{attribute 'linkalways'} 
{attribute 'no_explicit_call' := 'This FB is a CLASS and must be accessed using methods or properties'}
{attribute 'enable_dynamic_creation'}
FUNCTION_BLOCK _TcVnArray4_Point2_REAL EXTENDS AliasDatatypeBase
VAR
	localData : TcVnArray4_Point2_REAL;
	activeData : REFERENCE TO TcVnArray4_Point2_REAL REF= localData;
	aliasBaseDatatype : _Array0to3OfTcVnPoint2_REAL;
END_VAR

PROPERTY PUBLIC Address : PVOID
GET
Address := ADR(activeData);
END_GET
END_PROPERTY

METHOD PUBLIC ClearReference
VAR_INPUT
END_VAR
activeData REF= localData;
SetBaseDatatypeReference();
END_METHOD

METHOD PUBLIC Clone : I_Datatype
VAR
    pClone : POINTER TO _TcVnArray4_Point2_REAL;
END_VAR
pClone := __NEW(_TcVnArray4_Point2_REAL);
Clone := pClone^;
END_METHOD

METHOD FB_init : BOOL
VAR_INPUT
	bInitRetains : BOOL; // if TRUE, the retain variables are initialized (warm start / cold start)
	bInCopyCode : BOOL;  // if TRUE, the instance afterwards gets moved into the copy code (online change)
	//InitialValue : TcVnArray4_LREAL; // if possible, not all values can be initialized
END_VAR
//localData := InitialValue; // if possible, not all values can be initialized
SetBaseDatatypeReference();
AddBaseDatatype(aliasBaseDatatype);
END_METHOD

PROPERTY PUBLIC Identifier : T_MAXSTRING
GET
Identifier := 'TcVnArray4_Point2_REAL';
END_GET
END_PROPERTY

METHOD PUBLIC MakeReferenceTo
VAR_INPUT
	ReferenceTarget : REFERENCE TO TcVnArray4_Point2_REAL;
END_VAR
activeData REF= ReferenceTarget;
SetBaseDatatypeReference();
END_METHOD

METHOD PROTECTED SetBaseDatatypeReference
VAR_INPUT
END_VAR
aliasBaseDatatype.MakeReferenceTo(activeData);
END_METHOD

PROPERTY PUBLIC Size : UDINT
GET
Size := SIZEOF(activeData);
END_GET
END_PROPERTY

METHOD TryMakeReferenceTo : BOOL
VAR_INPUT
	Target : I_Datatype;
END_VAR
VAR
	pTargetData : POINTER TO TcVnArray4_Point2_REAL;
END_VAR
IF NOT IsEquivalentTo(Target) THEN
	RETURN;
END_IF

pTargetData := Target.Address;
activeData REF= pTargetData^;
SetBaseDatatypeReference();
TryMakeReferenceTo := TRUE;
END_METHOD

PROPERTY PUBLIC Value : REFERENCE TO TcVnArray4_Point2_REAL
GET
Value REF= activeData;
END_GET
END_PROPERTY

END_FUNCTION_BLOCK

(* stored: Version 1.1.0.1, ProductVersion 3.1.4024.13
   POU _TcVnArray4_Point2_REAL: Id {4025545f-dcd8-07f1-1107-87b0a050a007}, SpecialFunc None
   Folder Core: Id {1c224fdd-c286-067e-04f2-d6bc7c35533d}
   Folder Protected: Id {4b953cbc-0aa4-0180-3702-b88e6c1fe404}
   Folder Customize: Id {2d5a0047-d894-0c0c-1809-63d4316bbc29}
   Folder Constructor: Id {300c001e-6c28-0191-2240-26d28b2c7c34}
   Property Address: Id {fc659714-5bc5-0c7c-387d-10f77cbd39fe}
   Get Get: Id {d3ed5257-1d97-0b2d-1f86-5ac107c9d8f9}
   Method ClearReference: Id {282ccc3b-dbad-0830-2569-5c5e0bd79fea}
   Method Clone: Id {c3c1805b-f6b4-0162-321b-9fd4d2ee7ef1}
   Method FB_init: Id {7e656011-61f9-001c-3cc3-15cd8dc4d22e}
   Property Identifier: Id {87984a0e-07fe-0af7-3a9f-af2a916713fd}
   Get Get: Id {f0e7879e-9d2b-0d16-28fd-4b66622ea7b0}
   Method MakeReferenceTo: Id {98e70e59-24b5-08db-26f2-2157bb9f284f}
   Method SetBaseDatatypeReference: Id {eae12408-f2fd-0839-149b-9bf056c004f7}
   Property Size: Id {2a4b30d9-3b0c-0a29-3cfc-36c3efcd9243}
   Get Get: Id {8e2776be-6750-09fe-38b0-799294dd162a}
   Method TryMakeReferenceTo: Id {1e222f59-0c3e-046e-1f79-b4bdb77e13b8}
   Property Value: Id {8b8f4009-bb79-0b67-2c0c-473a8df55601}
   Get Get: Id {bc4bd116-2098-04e9-19a2-fac9cf2ea9af} *)
